FUNCTION_BLOCK OC_DONE_HMI (* Service Interface Function Block Type *)
  (* Standard: 61499-2 *)
  (* Version 0.0, 7/10/2026, Schneider Electric, template *)
  PACKAGE SE.Nereda;
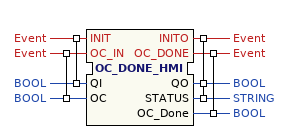
  EVENT_INPUT
    INIT WITH QI;
    OC_IN WITH OC;
  END_EVENT
  EVENT_OUTPUT
    INITO WITH QO, STATUS;
    OC_DONE WITH OC_Done;
  END_EVENT
  VAR_INPUT
    QI : BOOL;
    OC : BOOL;
  END_VAR
  VAR_OUTPUT
    QO : BOOL; (* Event Output Qualifier *)
    STATUS : STRING; (* Service Status *)
    OC_Done : BOOL;
  END_VAR
  SERVICE /
    SEQUENCE 
    END_SEQUENCE
  END_SERVICE
END_FUNCTION_BLOCK
